FUNCTION_BLOCK fb_EdgeDetector
VAR_INPUT
	bSignal			:	BOOL;
	timeON			:	TIME := T#200MS;
END_VAR
VAR_OUTPUT
	bRisingEdge		:	BOOL;
	bFallingEdge	: 	BOOL;
END_VAR
VAR
	timer			:	TON;
	bOnMeasure		:	BOOL;
	bOldState		: 	BOOL;
END_VAR

// set default state
timer.IN 	:= TRUE;
bRisingEdge	:= FALSE;
bFallingEdge:= FALSE;
timer.PT	:= timeON;
IF bSignal THEN
	IF NOT bSignal =  bOldState THEN
		// State wechsel
		timer.IN := FALSE;
		bOnMeasure := TRUE;
	END_IF
	IF timer.Q AND bOnMeasure THEN
		bOnMeasure := FALSE;
		bRisingEdge := TRUE;
	END_IF
ELSE
	IF NOT bSignal =  bOldState THEN
		// State wechsle
		timer.IN := FALSE;
		bOnMeasure := TRUE;
	END_IF
	IF timer.Q AND bOnMeasure THEN
		bOnMeasure := FALSE;
		bFallingEdge := TRUE;
	END_IF
END_IF

timer();

END_FUNCTION_BLOCK

(* stored: Version 1.1.0.1, ProductVersion 3.1.4024.12
   POU fb_EdgeDetector: Id {faa96c68-9e8b-4c42-b790-932233c76990}, SpecialFunc None *)
